// Mitsubishi GX Works2 project: 機電進階變異形連桿機構模組-ST   PLC: FX3U/FX3UC

// task Task_01 (event TRUE, interval 0, priority 31): POU_01

PROGRAM POU_01
VAR
  wEncoderPos : INT;
  wProgramStep : INT;
  bM2 : BOOL;
  wMaterialType : INT;
  tdT22 : TON;
  tdT0 : TON;
  tdT1 : TON;
  tdT28 : TON;
  wOrgPos : INT;
  wOffset : INT;
  bNoHMI : BOOL;
  bHigher : BOOL;
  tdT23 : TON;
  bM121 : BOOL;
  bM0 : BOOL;
  bM1 : BOOL;
  bM119 : BOOL;
  bM120 : BOOL;
  tdT100 : TON;
  tdT101 : TON;
END_VAR
(*
    Author: Steven Luo
    Date: 2018/10/16
*)

IF M8002 OR NOT X2 THEN
	wProgramStep := 0;
	ZRST(TRUE, Y0, Y17);
	bM0 := FALSE; (* 待機狀態 *)
	bM1 := FALSE; (* 運轉狀態 *)
	bM2 := FALSE;
	bM121 := FALSE;
	(* Configuration of FX2N-1HC *)
	TO(TRUE, K3, K0, K0, K1); (* Counter mode: 2-phase input, 2 edge count, 16 bits *)
END_IF;

(* Reading data from FX2N-2AD *)
TO(TRUE, H0, K1, K17, K1);
TO(TRUE, H2, K1, K17, K1);
FROM(TRUE, K1, K0, K2, K2M200);
D100 := K3M200;

(* Reading data from FX2N-1HC *)
TO(TRUE, H1, K0, K4, K1); (* Command: Count permit *)
FROM(TRUE, K0, K20, K1, D120); (* BFM #20, #21: Counter current value *)
wEncoderPos := D120;

IF bM0 AND M131 THEN (* HMI啟動 *)
	bM1 := TRUE;
END_IF;

IF M133 THEN (* HMI停止 *)
	bM1 := FALSE;
END_IF;

IF NOT X2 OR M140 THEN (* 按下急停 *)
	bM2 := TRUE;
END_IF;

IF (X2 OR NOT M140) AND bM2 THEN (* 放開急停，等待復歸 *)
	wProgramStep := 121;
END_IF;

IF M8002 THEN
	wProgramStep := 21;
	D211 := 1; D212 := 2; D213 := 3; D214 := 4; D215 := 5; D216 := 6; (* 出料位置 *)
	IF D201 = 0 THEN
		D201 := 420; (* 斜坡一位置 *)
	END_IF;
	IF D202 = 0 THEN
		D202 := 600; (* 斜坡二位置 *)
	END_IF;
	IF D203 = 0 THEN
		D203 := 780; (* 斜坡三位置 *)
	END_IF;
END_IF;

IF bM121 THEN (* 黃燈閃爍 *)
	tdT100(IN := NOT tdT101.Q, PT := T#500ms);
	tdT101(IN := tdT100.Q, PT := T#500ms);
	M143 := tdT100.Q;
ELSE
	RST(TRUE, M143);
END_IF;

IF M8002 OR M150 THEN
	D20 := 0; D21 := 0; D22 := 0; D23 := 0; D24 := 0; D25 := 0; D26 := 0; (* 進料數量 *)
END_IF;

IF bM0 AND NOT bM1 THEN (* 待機模式 *)
	M142 := TRUE; (* 綠燈亮 *)
	M144 := FALSE; (* 紅燈滅 *)
ELSE
	M142 := FALSE; (* 綠燈滅 *)
	M144 := TRUE; (* 紅燈亮 *)
END_IF;

IF M130 THEN (* 手動操作 *)
	IF M110 THEN (* 輸送帶正轉 *)
		Y0 := TRUE;
	ELSE
		Y0 := FALSE;
	END_IF;

	IF M111 THEN (* 輸送帶反轉 *)
		Y1 := TRUE;
	ELSE
		Y1 := FALSE;
	END_IF;

	IF M112 THEN (* 滑台左移 *)
		Y2 := TRUE;
	ELSE
		Y2 := FALSE;
	END_IF;

	IF M113 AND NOT X5 THEN (* 滑台右移 *)
		Y3 := TRUE;
	ELSE
		Y3 := FALSE;
	END_IF;

	IF M114 THEN (* 垂直缸下降 *)
		Y4 := TRUE;
	END_IF;

	IF M115 THEN (* 垂直缸上升 *)
		Y4 := FALSE;
	END_IF;

	IF X11 AND M116 THEN (* 水平缸前進 *)
		Y5 := TRUE;
	ELSE
		Y5 := FALSE;
	END_IF;

	IF X11 AND M117 THEN (* 水平缸後退 *)
		Y6 := TRUE;
	ELSE
		Y6 := FALSE;
	END_IF;

	IF M118 THEN (* 吸盤吸 *)
		tdT1(IN := FALSE);
		Y10 := FALSE;
		Y7 := TRUE;
	END_IF;

	IF M119 THEN (* 吸盤放 *)
		Y7 := FALSE;
		Y10 := TRUE;
	ELSE
		Y10 := FALSE;
	END_IF;

	IF M120 THEN (* 滑台回原點 *)
		IF NOT X5 THEN
			bM120 := TRUE;
		END_IF;
	END_IF;
	IF bM120 AND NOT X5 THEN
		Y3 := TRUE;
	ELSE
		IF X5 THEN
			Y3 := FALSE;
			bM120 := FALSE;
		END_IF;
	END_IF;
	
	IF M151 THEN (* 斜坡一位置 *)
		D201 := D120;
	END_IF;
	IF M152 THEN (* 斜坡二位置 *)
		D202 := D120;
	END_IF;
	IF M153 THEN (* 斜坡三位置 *)
		D203 := D120;
	END_IF;
END_IF; (* 手動操作 *)

IF (D211 = D212) OR (D211 = D213) OR (D211 = D214) OR (D211 = D215) OR (D211 = D216) THEN
	M191 := TRUE;
ELSE
	M191 := FALSE;
END_IF;

IF (D212 = D211) OR (D212 = D213) OR (D212 = D214) OR (D212 = D215) OR (D212 = D216) THEN
	M192 := TRUE;
ELSE
	M192 := FALSE;
END_IF;

IF (D213 = D212) OR (D211 = D213) OR (D213 = D214) OR (D213 = D215) OR (D213 = D216) THEN
	M193 := TRUE;
ELSE
	M193 := FALSE;
END_IF;

IF (D214 = D212) OR (D214 = D213) OR (D211 = D214) OR (D214 = D215) OR (D214 = D216) THEN
	M194 := TRUE;
ELSE
	M194 := FALSE;
END_IF;

IF (D215 = D212) OR (D215 = D213) OR (D215 = D214) OR (D211 = D215) OR (D215 = D216) THEN
	M195 := TRUE;
ELSE
	M195 := FALSE;
END_IF;

IF (D216 = D212) OR (D216 = D213) OR (D216 = D214) OR (D216 = D215) OR (D211 = D216) THEN
	M196 := TRUE;
ELSE
	M196 := FALSE;
END_IF;

CASE wProgramStep OF
	21:
		IF X5 AND X11 AND X13 AND NOT X15 THEN (* 原點條件: 編碼器在原點，垂直缸在上位，水平缸縮回，吸盤放 *)
			bNoHMI := FALSE;
			bM0 := TRUE;
			bM1 := FALSE;
			bM121 := FALSE;
			IF X0 OR M131 THEN (* 工作模式、按下啟動鈕 *)
				tdT0(IN := FALSE);
				tdT22(IN := FALSE);
				tdT23(IN := FALSE);
				tdT28(IN := FALSE);
				IF X0 THEN
					bNoHMI := TRUE;
				END_IF;
				wProgramStep := 22;
			END_IF;
		END_IF;
	22:
		bM0 := FALSE;
		D0 := 0;
		tdT1(IN := FALSE);
		bHigher := FALSE;
		wMaterialType := 0;
		Y0 := TRUE; (* 輸送帶前進 *)
		tdT0(IN := TRUE, PT := T#10s); (* 計時10秒 *)
		IF NOT X3 AND X4 THEN (* 塑料、藍色 *)
			wMaterialType := 1;
		ELSIF X3 AND X4 THEN (* 金屬、銀色 *)
			wMaterialType := 2;
		ELSIF X3 AND NOT X4 THEN (* 金屬、黑色 *)
			wMaterialType := 3;
		END_IF;
		IF wMaterialType > 0 THEN
			tdT22(IN := TRUE, PT := T#500ms);
		END_IF;
		IF tdT0.Q AND wMaterialType = 0 THEN (* 無料 *)
			Y0 := FALSE; (* 輸送帶停止 *)
			bM1 := FALSE;
			wProgramStep := 21;
		END_IF;
		IF tdT22.Q THEN
			Y0 := FALSE; (* 輸送帶停止 *)
			wProgramStep := 23;
			D20 := D20 + 1;
		END_IF;
	23:
		Y4 := TRUE; (* 垂直缸下降 *)
		IF X12 THEN
			tdT23(IN := TRUE, PT := T#1s);
			IF tdT23.Q THEN
				IF D100 > WORD_TO_INT(K2400) THEN
					bHigher := TRUE; (* 高料 *)
				END_IF;
				Y7 := TRUE; (* 吸盤吸 *)
				IF X15 THEN
					IF NOT bNoHMI THEN;
						IF NOT bHigher THEN
							wMaterialType := wMaterialType + 3;
						END_IF;
						D0 := wMaterialType;
						CASE D0 OF
						1:
							D21 := D21 + 1;
						2:
							D22 := D22 + 1;
						3:
							D23 := D23 + 1;
						4:
							D24 := D24 + 1;
						5:
							D25 := D25 + 1;
						6:
							D26 := D26 + 1;
						END_CASE;
					END_IF;
					Y4 := FALSE; (* 垂直缸上升 *)
					wProgramStep := 24;
				END_IF;
			END_IF;
		END_IF;
	24:
		IF X11 THEN
			wOrgPos := wEncoderPos;
			Y2 := TRUE; (* 滑台前進 *)
			wProgramStep := 25;
		END_IF;
	25:
		wOffset := wEncoderPos - wOrgPos;
		IF bNoHMI THEN
			IF (wMaterialType = 1) AND (wOffset >= 800 AND wOffset < 1170) THEN (* 第一格 *)
				Y2 := FALSE;
			ELSIF (wMaterialType = 2) AND (wOffset >= 1170 AND wOffset <1540 ) THEN (* 第二格 *)
				Y2 := FALSE;
			ELSIF (wMaterialType = 3) AND (wOffset >= 1540) THEN (* 第三格 *)
				Y2 := FALSE;
			END_IF;
		ELSE
			IF (wOffset >= D201 AND wOffset < D202) THEN (* 第一格 *)
				IF (wMaterialType = D211) OR (wMaterialType = D214) THEN
					Y2 := FALSE;
				END_IF;
			ELSIF (wOffset >= D202 AND wOffset < D203 ) THEN (* 第二格 *)
				IF (wMaterialType = D212) OR (wMaterialType = D215) THEN
					Y2 := FALSE;
				END_IF;
			ELSIF (wOffset >= D203) THEN (* 第三格 *)
				IF (wMaterialType = D213) OR (wMaterialType = D216) THEN
					Y2 := FALSE;
				END_IF;
			END_IF;
		END_IF;
		IF NOT Y2 THEN
			wProgramStep := 26;
		END_IF;
	26:
		IF bNoHMI THEN
			IF bHigher THEN (* 高料放上層 *)
				Y5 := TRUE; (* 水平缸前進 *)
				IF X14 THEN
					Y5 := FALSE;
					wProgramStep := 28;
				END_IF;
			ELSE (* 低料放下層 *)
				wProgramStep := 27;
			END_IF;
		ELSE
			IF (wMaterialType = D211) OR (wMaterialType = D212) OR (wMaterialType = D213) THEN (* 上層 *)
				Y5 := TRUE; (* 水平缸前進 *)
				IF X14 THEN
					Y5 := FALSE;
					wProgramStep := 28;
				END_IF;
			ELSIF (wMaterialType = D214) OR (wMaterialType = D215) OR (wMaterialType = D216) THEN (* 下層 *)
				wProgramStep := 27;
			END_IF;
		END_IF;
	27:
		Y4 := TRUE; (* 垂直缸下降 *)
		IF X12 THEN
			wProgramStep := 28;
		END_IF;
	28:
		Y7 := FALSE;
		Y10 := TRUE; (* 吸盤放開 *)
		tdT28(IN := TRUE, PT := T#500ms);
		IF tdT28.Q THEN
			Y10 := FALSE;
			IF bNoHMI THEN
				IF bHigher THEN (* 高料 *)
					wProgramStep := 30;
				ELSE (* 低料 *)
					wProgramStep := 29;
				END_IF;
			ELSE
				IF (wMaterialType = D211) OR (wMaterialType = D212) OR (wMaterialType = D213) THEN (* 上層 *)
					wProgramStep := 30;
				ELSIF (wMaterialType = D214) OR (wMaterialType = D215) OR (wMaterialType = D216) THEN (* 下層 *)
					wProgramStep := 29;
				END_IF;
			END_IF;
		END_IF;
	29:
		Y4 := FALSE; (* 垂直缸上升 *)
		IF X11 THEN
			wProgramStep := 31;
		END_IF;
	30:
		Y6 := TRUE; (* 水平缸後退 *)
		IF X13 THEN
			Y6 := FALSE;
			wProgramStep := 31;
		END_IF;
	31:
		Y3 := TRUE; (* 滑台後退 *)
		IF X5 THEN
			tdT1(IN := TRUE, PT := T#100ms);
			IF tdT1.Q THEN
				Y3 := FALSE;
				IF bNoHMI THEN
					IF X1 THEN (* 連續循環 *)
						IF bM121 THEN
							wProgramStep := 21;
						ELSE
							tdT0(IN := FALSE);
							tdT22(IN := FALSE);
							tdT23(IN := FALSE);
							tdT28(IN := FALSE);
							wProgramStep := 22;
						END_IF;
					ELSE (* 單一循環 *)
						wProgramStep := 21;
					END_IF;
				ELSE
					IF M130 THEN (* 手動 *)
						wProgramStep := 21;
					ELSE (* 自動 *)
						IF bM121 OR NOT bM1 THEN
							wProgramStep := 21;
						ELSE
							tdT0(IN := FALSE);
							tdT22(IN := FALSE);
							tdT23(IN := FALSE);
							tdT28(IN := FALSE);
							wProgramStep := 22;
						END_IF;
					END_IF;
				END_IF; (* bNoHMI *)
			END_IF; (* tdT1.Q *)
		END_IF; (* X5 *)
	121:
		IF X0 OR M132 THEN (* 復歸模式、按下啟動鈕 *)
			bM2 := FALSE;
			bM121 := TRUE;
			wProgramStep := 28;
		END_IF;
	ELSE
	;
END_CASE;
END_PROGRAM
